(* CoDeSys 2.3 export: STE.EXP *)

(* Data type in BathFB *)
TYPE StE :
(
    on,
    off1,
    not_enabled
);
END_TYPE
